FUNCTION_BLOCK FB_HINNAN_ARPOMINEN
VAR_INPUT
END_VAR
VAR_OUTPUT
	arrPrices:				ARRAY[1..96] OF REAL;	//Arvot
END_VAR
VAR
	i:						INT;
	nRange:					DINT :=10000;			//Vaihteluväli
	frand:					Drand;
	fPrice:					REAL;
	fValue:					DINT;
END_VAR

FOR i := 1 TO 96 DO
frand();
fValue:= LREAL_TO_DINT (fRand.num*nRange);
fPrice:= DINT_TO_REAL (fValue)/1000; 
arrPrices[i] := fPrice;
END_FOR

END_FUNCTION_BLOCK

(* stored: Version 1.1.0.1
   POU FB_HINNAN_ARPOMINEN: Id {35ed4ceb-fdb2-4e75-8a54-fe23768ff27a}, SpecialFunc None *)
